PROGRAM POU_MINUS
VAR
	Result:REAL;
	Value01:REAL;
	Value02:REAL;
END_VAR

Result:=MAIN.Value01-MAIN.Value02;

END_PROGRAM

(* stored: Version 1.1.0.1, ProductVersion 3.1.4024.4
   POU POU_MINUS: Id {c9ff0511-ce0d-4cd8-aec9-8b7f3711ba7e}, SpecialFunc None *)
